FUNCTION_BLOCK Mc3MoveRelativeTask EXTENDS Mc3MotionTask
VAR
	_TargetDistance : LREAL;
	McMoveRelative	: ARRAY[0..1] OF Tc3_Mc3Ptp.MC_MoveRelative;
	Active			: UDINT;
    _McBufferMode	: Tc3_Mc3Ptp.EBufferMode;
END_VAR

PROPERTY BufferMode : REFERENCE TO Tc3_Mc3Ptp.EBufferMode
GET
BufferMode REF= _McBufferMode;
END_GET
END_PROPERTY

{attribute 'monitoring' := 'call'}
PROPERTY Busy : BOOL
GET
Busy := McMoveRelative[Active].Busy;
END_GET
END_PROPERTY

METHOD CyclicLogic
VAR
    i : UDINT;
END_VAR
FOR i := 0 TO 1 DO
	McMoveRelative[i](Axis		   := _Axis.Axis,
					  Distance	   := _TargetDistance,
					  Velocity	   := _Axis.Velocity,
					  Acceleration := _Axis.Acceleration,
					  Deceleration := _Axis.Deceleration,
					  Jerk		   := _Axis.Jerk,
					  BufferMode   := _McBufferMode);

	McMoveRelative[i].Execute := FALSE;
END_FOR
END_METHOD

{attribute 'monitoring' := 'call'}
PROPERTY Error : BOOL
GET
Error := McMoveRelative[Active].Error;
END_GET
END_PROPERTY

{attribute 'monitoring' := 'call'}
PROPERTY ErrorId : UDINT
GET
ErrorID := McMoveRelative[Active].ErrorID;
END_GET
END_PROPERTY

METHOD Execute : BOOL;
IF Active = 0 THEN
	Active := 1;
	McMoveRelative[Active](Axis			:= _Axis.Axis,
						   Execute		:= TRUE,
						   Distance		:= _TargetDistance,
						   Velocity		:= _Axis.Velocity,
						   Acceleration := _Axis.Acceleration,
						   Deceleration := _Axis.Deceleration,
						   Jerk			:= _Axis.Jerk,
						   BufferMode	:= _McBufferMode);
ELSE
	Active := 0;
	McMoveRelative[Active](Axis			:= _Axis.Axis,
						   Execute		:= TRUE,
						   Distance		:= _TargetDistance,
						   Velocity		:= _Axis.Velocity,
						   Acceleration := _Axis.Acceleration,
						   Deceleration := _Axis.Deceleration,
						   Jerk			:= _Axis.Jerk,
						   BufferMode	:= _McBufferMode);
END_IF

Execute := TRUE;
END_METHOD

{attribute 'monitoring' := 'call'}
PROPERTY TargetDistance : LREAL
SET
_TargetDistance := TargetDistance;
END_SET
END_PROPERTY

END_FUNCTION_BLOCK

(* stored: Version 1.1.0.1, ProductVersion 3.1.4026.20
   POU Mc3MoveRelativeTask: Id {747564a4-0c65-4429-b7a7-317eab0d9d62}, SpecialFunc None
   Property BufferMode: Id {cf6af077-c467-4459-98e8-05335da0940f}
   Get Get: Id {d37a5b63-be04-4ae1-8719-21a7a111e319}
   Property Busy: Id {5d4330f2-e64a-4de5-b48d-004294a79bb7}
   Get Get: Id {c18237b4-3a61-4e79-bc45-2ed4e922e456}
   Method CyclicLogic: Id {f422cf3f-402d-410e-9eb3-c26e5cc02780}
   Property Error: Id {8e1cf5c6-2c3f-4052-9585-3184d387e1f7}
   Get Get: Id {7a8d35b3-9c80-4747-afa2-3b6c31517e34}
   Property ErrorId: Id {ce6bb234-f6e3-4271-895c-20e6ff8650ad}
   Get Get: Id {0e762977-7f5f-43d0-808f-8c2a3aac8e5d}
   Method Execute: Id {db9ca5b3-a0ca-43f1-ab12-88b704590577}
   Property TargetDistance: Id {5a06b370-fc7b-47e4-ac8f-01725796dc66}
   Set Set: Id {69b37b4c-ebca-4b16-9d7d-723a280393e3} *)
